(* IEC 61131-3 sources: CodesysTest/alpha/export/FBs/DelayDwellFB/DelayDwellFB.pou/DelaySetting.prop, 1 file *)

(* ---- Set.pm.st ---- *)
(*#-#-#-#-#-#-#-#-#-#---Declaration---#-#-#-#-#-#-#-#-#-#-#-#-#*)

VAR
END_VAR
(*#-#-#-#-#-#-#-#-#-#---Implementation---#-#-#-#-#-#-#-#-#-#-#-#-#*)

_delayTimeInMS := DelaySetting;
